// TIA Portal V16 export
// export: Created 2022-09-01T13:36:50.3452127Z, ExportSetting WithDefaults, DisplayName Totally Integrated Automation Portal, DisplayVersion V16, DisplayName TIA Portal Version Control Interface, DisplayVersion V16, DisplayName TIA Portal Openness, DisplayVersion V16, DisplayName STEP 7 Professional, DisplayVersion V16, DisplayName STEP 7 Safety, DisplayVersion V16, DisplayName WinCC Advanced, DisplayVersion V16
DATA_BLOCK "Níveis_TK02_TK03"   // DB11
{ S7_Optimized_Access := 'TRUE' }
VERSION : 0.1
// stored: AutoNumber true, IsOnlyStoredInLoadMemory false, IsRetainMemResEnabled false, IsWriteProtectedInAS false, MemoryReserve 100
   VAR
      LSH301 : Bool;
      LSM301 : Bool;
   END_VAR
   VAR RETAIN
      LSL301 : Bool;
   END_VAR
   VAR
      LSH201 : Bool;
      LSM201 : Bool;
      LSL201 : Bool;
      NÍVEL_EM_METROS_TK03 : Real;
      NÍVEL_EM_METROS_TK02 : Real;
   END_VAR
BEGIN
END_DATA_BLOCK
